(* IEC 61131-3 sources: modbus_udp_test/test_2/applications/Core_1_3_2/Регуляторы, 1 file *)

(* ---- REGULATOR.PRG ---- *)
PROGRAM REGULATOR
VAR
	pid_control		:	pid_control;
END_VAR

// === IMPLEMENTATION ===

pid_control();
